TYPE ST_VALID_OBSERVERS :
STRUCT
	cnt:		INT;
	observers:	ARRAY[0..GVL_GENERIC_OBSERVER.OBSERVER_CNT-1] OF ST_GENERIC_OBSERVER;
END_STRUCT
END_TYPE

(* stored: Version 1.1.0.1, ProductVersion 3.1.4026.18
   DUT ST_VALID_OBSERVERS: Id {b0554414-3548-460f-b8f9-696f12abc41b} *)
